# EPICS IOC start-up script: iocsh/ethercatmcAnalogInputSmooAdelMdel.iocsh
ethercatmcCreateAsynParam $(MOTOR_PORT) $(ASYNPARAMNAME)      Float64

<<<<<<< HEAD
dbLoadRecords("ethercatmcAnalogInput.template", "P=$(P), R=$(R), MOTOR_PORT=$(MOTOR_PORT), CHNO=$(CHNO), ASYNPARAMNAME=$(ASYNPARAMNAME), PREC=$(PREC), DESC=$(DESC), EGU=$(EGU), SMOO=$(SMOO), ADEL=$(ADEL), MDEL=$(MDEL)")
=======
dbLoadRecords("ethercatmcAnalogInputSmooAdelMdel.template", "P=$(P), R=$(R), MOTOR_PORT=$(MOTOR_PORT), CHNO=$(CHNO), ASYNPARAMNAME=$(ASYNPARAMNAME), PREC=$(PREC), DESC=$(DESC), EGU=$(EGU), SMOO=$(SMOO), ADEL=$(ADEL), MDEL=$(MDEL)")
>>>>>>> github/master
